INTERFACE ITF_TopElement1 EXTENDS ITF_BaseTopElement

END_INTERFACE

(* stored: Version 1.1.0.1, ProductVersion 3.1.4024.15
   Itf ITF_TopElement1: Id {bf8e1ef0-d5d2-4ec0-8036-295070c74954} *)
